// Mitsubishi GX Works2 project: De09   PLC: FX2N/FX2NC

PROGRAM MAIN
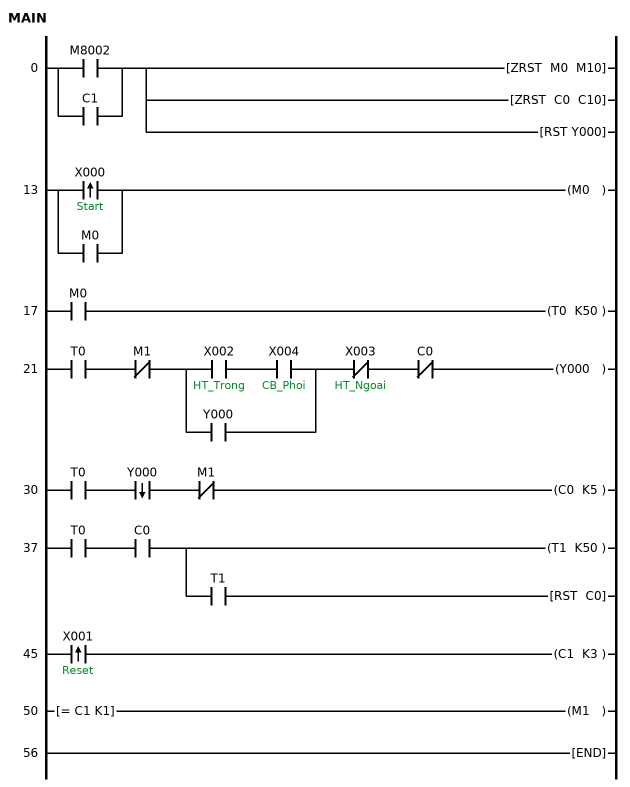
0     LD      M8002
      OR      C1
      ZRST    M0 M10
      ZRST    C0 C10
      RST     Y000
13    LDP     X000  ; Start
      OR      M0
      OUT     M0
17    LD      M0
      OUT     T0 K50
21    LD      T0
      ANI     M1
      LD      X002  ; HT_Trong
      AND     X004  ; CB_Phoi
      OR      Y000
      ANB
      ANI     X003  ; HT_Ngoai
      ANI     C0
      OUT     Y000
30    LD      T0
      ANDF    Y000
      ANI     M1
      OUT     C0 K5
37    LD      T0
      AND     C0
      OUT     T1 K50
      AND     T1
      RST     C0
45    LDP     X001  ; Reset
      OUT     C1 K3
50    LD=     C1 K1
      OUT     M1
56    END
END_PROGRAM
